Staubli VAL3: JointVel.dtx

public num jv[6]
